{attribute 'linkalways'} 
{attribute 'no_explicit_call' := 'This FB is a CLASS and must be accessed using methods or properties'}
{attribute 'enable_dynamic_creation'}
FUNCTION_BLOCK Node_F_VN_GetImageInfo EXTENDS Node
VAR
    ipImage : _ITcVnImage;
    stImageInfo : _TcVnImageInfo;
    hrPrev : _HRESULT(S_OK);
	hresult : _HRESULT(S_OK);
END_VAR

METHOD PUBLIC  Clone : I_Node
VAR
	pNode : POINTER TO Node_F_VN_GetImageInfo;
END_VAR
pNode := __NEW(Node_F_VN_GetImageInfo);
Clone := pNode^;
END_METHOD

METHOD FB_init : BOOL
VAR_INPUT
	bInitRetains : BOOL; // if TRUE, the retain variables are initialized (warm start / cold start)
	bInCopyCode : BOOL;  // if TRUE, the instance afterwards gets moved into the copy code (online change)
END_VAR
AddInput('ipImage', ipImage);
AddInput('hrPrev', hrPrev);
AddOutput('stImageInfo', stImageInfo);
AddOutput('hresult',hresult);
END_METHOD

METHOD PROTECTED OnExecute : HRESULT
hresult.Value := F_VN_GetImageInfo(
    ipImage := ipImage.Value,
	stImageInfo := stImageInfo.Value,
	hrPrev:= hrPrev.Value);
END_METHOD

END_FUNCTION_BLOCK

(* stored: Version 1.1.0.1, ProductVersion 3.1.4024.13
   POU Node_F_VN_GetImageInfo: Id {973cae40-1586-09c8-2150-b768b5b07f6e}, SpecialFunc None
   Folder Constructor: Id {e319145f-f582-0a7b-173a-c1cce6523e52}
   Method Clone: Id {662662af-1580-0668-1f61-1dee41ffec85}
   Method FB_init: Id {7121d6e6-127e-0e81-137c-824cbfd5d89c}
   Method OnExecute: Id {ae41b3a6-0634-0c28-0d4f-55a9cf780d4f} *)
